VAR_GLOBAL
	{attribute 'OPC.UA.DA' := '1'}
	{attribute 'OPC.UA.DA.Description' := 'Methods with different InputOutput types'} 	
	Methods : FB_Methods;
	
	{attribute 'OPC.UA.DA' := '1'}
	{attribute 'OPC.UA.DA.Description' := 'Methods with mathematical functions'}
	Mathematics : FB_Mathematics;

	{attribute 'OPC.UA.DA' := '1'}
	{attribute 'OPC.UA.DA.Description' := 'Job method which execution may take longer than a PLC cycle'}
	Job : FB_Job;	
END_VAR

(* stored: Version 1.1.0.1, ProductVersion 3.1.4024.11
   GVL GVL_methods: Id {ed212e00-68d5-48e7-8c2d-6f495f9062bb} *)
